INTERFACE IHandling EXTENDS ZApplication.IUnit

END_INTERFACE

(* stored: Version 1.1.0.1
   Itf IHandling: Id {f2a4b17f-26f2-4bad-91fb-18d923adeba3} *)
